FUNCTION_BLOCK StringQueue EXTENDS Queue
VAR
	elements : FB_BA_DynamicArray := (uiEntrySize := SIZEOF(STRING), uiMinExpCount := CONSTS.initArraySize);
	//length : USINT := 0;
END_VAR

METHOD get : STRING
VAR_INPUT
	i : UINT;
END_VAR
elements.GetEntry(diIndex := i, pResultEntry := ADR(get));
END_METHOD

METHOD isEmpty : BOOL
VAR_INPUT
END_VAR
isEmpty := (elements.diCount = 0);
END_METHOD

METHOD poll : STRING
VAR_INST
	temp : STRING;
	i : UINT;
END_VAR
temp := get(i := 0);
elements.RemoveEntry(diIndex := 0);
//length := length - 1;
poll := temp;
END_METHOD

METHOD push : BOOL
VAR_INPUT
	value : STRING;
END_VAR
elements.AddEntry(pEntry := ADR(value));
//length := length + 1;
END_METHOD

METHOD size : DINT
VAR_INPUT
END_VAR
size := elements.diCount;
END_METHOD

END_FUNCTION_BLOCK

(* stored: Version 1.1.0.1, ProductVersion 3.1.4024.11
   POU StringQueue: Id {d0805259-a10e-466f-82e5-5e0980abf977}, SpecialFunc None
   Method get: Id {f6e1b64e-ef1a-40af-815a-e4f7b939695e}
   Method isEmpty: Id {f02a231f-f5b4-4a0a-86be-fb8c5cd7be57}
   Method poll: Id {9f031a82-eb77-4afe-8554-88232cc2f2e6}
   Method push: Id {33102ce9-4361-45fb-9c60-c63261e6725b}
   Method size: Id {9a118a6a-ea85-40be-b672-dfdf0f839afb} *)
